PROGRAM MAIN
VAR
    _sampleContext : SampleContext;
END_VAR

_sampleContext.Run();

END_PROGRAM

(* stored: Version 1.1.0.1, ProductVersion 3.1.4024.9
   POU MAIN: Id {2b66492f-ba52-0f75-2e94-09654a948221}, SpecialFunc None *)
